PROGRAM Version
VAR
END_VAR

(*

1.0.1.1:	Boido	020120

Version.txt replaced with Version PRG

1.0.2.2:	Boido	020120

VersionLib removed.

*)

END_PROGRAM

(* stored: Version 1.1.0.1, ProductVersion 3.1.4024.0
   POU Version: Id {95618842-63da-482f-8530-b7fbf5f82af2}, SpecialFunc None *)
